INTERFACE I_HostGraphs

PROPERTY Graphs : I_Graphs
GET
END_GET
END_PROPERTY

END_INTERFACE

(* stored: Version 1.1.0.1, ProductVersion 3.1.4024.12
   Itf I_HostGraphs: Id {0ac488b4-54d0-4c12-951b-d9b20b69f03c}
   Property Graphs: Id {197e5d25-ba9a-43e7-a4b6-3950cb5aa040}
   Get Get: Id {3b5e175c-76af-4cff-899c-968aa8efffa9} *)
